INTERFACE I_Component

METHOD AddChild
VAR_INPUT
	Child : I_Component;
END_VAR
END_METHOD

METHOD GetChildren : ARRAY [1..Param.NumberOfChildren] OF I_Component;
END_METHOD

PROPERTY GetSize : INT
GET
END_GET
END_PROPERTY

END_INTERFACE

(* stored: Version 1.1.0.1, ProductVersion 3.1.4024.12
   Itf I_Component: Id {317cf77d-fe68-475e-9ce3-3fca36253e36}
   Method AddChild: Id {8380aa88-8fcd-4ff4-8451-dd079d5864ab}
   Method GetChildren: Id {9b5cbc35-a5f4-4729-9385-019e7b8b28a6}
   Property GetSize: Id {2f131b1a-ac03-4b6f-9ce3-d5855561434c}
   Get Get: Id {2bed0d92-cc0a-482a-bb6b-c91d420036f7} *)
